TYPE ST_RingBufferIOPart :
STRUCT
	(*200當確認點、是否傳送到*)
	Table	: ARRAY [0..200] OF BOOL;
END_STRUCT
END_TYPE

(* stored: Version 1.1.0.1, ProductVersion 3.1.4024.9
   DUT ST_RingBufferIOPart: Id {71d192d5-ba46-410f-8628-b87414470e18} *)
